// TwinCAT 3 PLC project PlcTc3JsonXmlSampleJsonDataType
// ProgramVersion: 3.1.4021.2
// libraries:
//   Tc2_Standard, * (Beckhoff Automation GmbH)
//   Tc2_System, * (Beckhoff Automation GmbH)
//   Tc3_JsonXml, * (Beckhoff Automation GmbH)
//   Tc3_Module, * (Beckhoff Automation GmbH)
// project tree:
//   DUTs/ ST_Values.TcDUT
//   / PlcTask.TcTTO
//   POUs/ MAIN.TcPOU
// real-time tasks:
//   TASK PlcTask: cycle T#10ms, priority 20, ADS port 350

CONFIGURATION PlcTc3JsonXmlSampleJsonDataType
    RESOURCE PLC ON TwinCAT3
        TASK PlcTask(INTERVAL := T#10ms, PRIORITY := 20);
        PROGRAM MAIN WITH PlcTask : MAIN;
    END_RESOURCE
END_CONFIGURATION

// ---- DUTs/ST_Values.TcDUT
TYPE ST_Values :
STRUCT
	  {attribute 'Unit' := 'm/s'}
	  {attribute 'DisplayName' := 'Speed'}
	  Sensor1   : REAL := 42.42;
	  {attribute 'Unit' := 'V'}
	  {attribute 'DisplayName' := 'Voltage'}
	  Sensor2	: DINT := 230;
	  {attribute 'Unit' := 'A'}
	  {attribute 'DisplayName' := 'Current'}
	  Sensor3	: DINT := 3;
END_STRUCT
END_TYPE

// ---- POUs/MAIN.TcPOU
PROGRAM MAIN
VAR
	dtTimestamp : DATE_AND_TIME := DT#2017-04-04-12:42:42;
  	(* JSON document *)
  	fbJson			: FB_JsonSaxWriter;
	fbJsonDataType	: FB_JsonReadWriteDataType;
	sJsonDoc		: STRING(255); // Small JSON document, can be generated via GetDocument() for up to 255 characters
	sJsonDoc2		: STRING(2000); // Large JSON document, can be generated via CopyDocument()
	stValues		: ST_Values;
END_VAR

fbJson.ResetDocument();
fbJson.StartObject();
fbjson.AddKeyDateTime('Timestamp', dtTimestamp);
fbJsonDataType.AddJsonKeyValueFromSymbol(fbJson, 'Values', 'ST_Values', SIZEOF(stValues), ADR(stValues));
fbJsonDataType.AddJsonKeyPropertiesFromSymbol(fbJson, 'MetaData', 'ST_Values', 'Unit|DisplayName');
fbJson.EndObject();

sJsonDoc := fbJson.GetDocument();
fbJson.CopyDocument(sJsonDoc2, SIZEOF(sJsonDoc2));

END_PROGRAM
